(* IEC 61131-3 sources: vertriebstagung/PLC_Kessel, 1 file *)

(* ---- PLC_PRG.st ---- *)
PROGRAM PLC_PRG
VAR
    myVar : INT := 5;
END_VAR

myVar := myVar + 1;

WHILE myVar > 10 DO
    ;
END_WHILE;

test(); /* changes on the devbranch only */

END_PROGRAM

ACTIONS
    ACTION test
        ;
    END_ACTION
END_ACTIONS
